// Mitsubishi GX Works2 project: 정수를 실수로   PLC: Q02/Q02H

PROGRAM MAIN
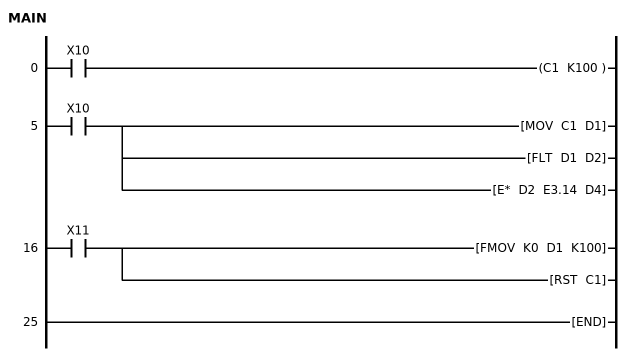
0     LD      X10
      OUT     C1 K100
5     LD      X10
      MOV     C1 D1
      FLT     D1 D2
      E*      D2 E3.14 D4
16    LD      X11
      FMOV    K0 D1 K100
      RST     C1
25    END
END_PROGRAM
